ABB RobotStudio station: ABBRacer_20170305-223939.rsstn

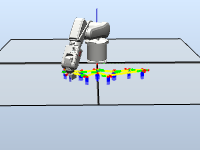
Station ABBRacer (saved by RobotStudio 6.4.7206.1027)
Controller IRB_120_3kg_0.58m, task T_ROB1: task frame (RAPID world) sits at (0, 0, 25) mm in the station
Controller IRB_120_3kg_0.58m
  mechanical unit ROB_1: IRB120_3_58__01, 6 joints, base frame (0, 0, 0) mm
Layout (positions relative to the parent item):
  - IRB120_3_58__01 [mechanism, from Robots\IRB120_3_58_G_01.rslib] at (0, 0, 25) mm; joint values [-0.4552, 1.5213, -0.5651, 0, 0.6146, 3.1228] (rad or m)
  - Bakje [part] at (432.53, -170.17, 50) mm, rotated rx -90 ry 0 rz 155 deg
Attachment: Bakje is attached to IRB120_3_58__01 / Link6
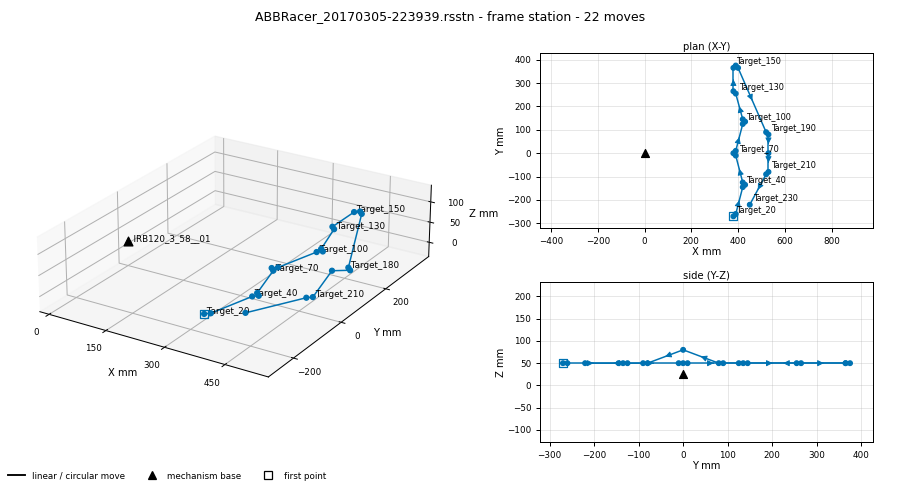
[picture p0: tool path of ABBRacer_20170305-223939.rsstn in frame station, 22 of 22 moves have a stored position in this frame; points joined in program order, loops and branches not executed]
Targets, tools, work objects and paths stored in the station, written as RAPID:
! task T_ROB1
MODULE Module1
  CONST robtarget Target_20:=[[380,-270,25],[0,0,1,0],[-1,0,-1,0],[9E+09,9E+09,9E+09,9E+09,9E+09,9E+09]];
  CONST robtarget Target_30:=[[390,-260,25],[0,0.130526192,0.991444861,0],[-1,-1,-1,0],[9E+09,9E+09,9E+09,9E+09,9E+09,9E+09]];
  CONST robtarget Target_40:=[[420,-145,25],[0,0.258819045,0.965925826,0],[-1,0,-1,0],[9E+09,9E+09,9E+09,9E+09,9E+09,9E+09]];
  CONST robtarget Target_50:=[[430.000232033,-134.999844259,25.000157187],[0.00000015,0,1,-0.000000047],[-1,0,-1,0],[9E+09,9E+09,9E+09,9E+09,9E+09,9E+09]];
  CONST robtarget Target_60:=[[420,-125,25],[0,-0.130526192,0.991444861,0],[-1,0,-1,0],[9E+09,9E+09,9E+09,9E+09,9E+09,9E+09]];
  CONST robtarget Target_70:=[[390,-10,25],[0,-0.3007058,0.953716951,0],[-1,-1,-1,0],[9E+09,9E+09,9E+09,9E+09,9E+09,9E+09]];
  CONST robtarget Target_80:=[[380.000012735,0,25.000038681],[0.000000135,0,1,0],[0,0,0,0],[9E+09,9E+09,9E+09,9E+09,9E+09,9E+09]];
  CONST robtarget Target_90:=[[390,10,25],[0,0.130526192,0.991444861,0],[0,0,0,0],[9E+09,9E+09,9E+09,9E+09,9E+09,9E+09]];
  CONST robtarget Target_100:=[[420,125,25],[0,0.3007058,0.953716951,0],[0,-1,0,0],[9E+09,9E+09,9E+09,9E+09,9E+09,9E+09]];
  CONST robtarget Target_110:=[[430,135,25],[0,0,1,0],[0,-1,0,0],[9E+09,9E+09,9E+09,9E+09,9E+09,9E+09]];
  CONST robtarget Target_120:=[[420,145,25],[0,-0.130526192,0.991444861,0],[0,-1,0,0],[9E+09,9E+09,9E+09,9E+09,9E+09,9E+09]];
  CONST robtarget Target_130:=[[390,255,25],[0,-0.3007058,0.953716951,0],[0,0,0,0],[9E+09,9E+09,9E+09,9E+09,9E+09,9E+09]];
  CONST robtarget Target_140:=[[379.999778696,265.000063835,24.999829243],[-0.000000287,0,1,-0.0000002],[0,0,0,0],[9E+09,9E+09,9E+09,9E+09,9E+09,9E+09]];
  CONST robtarget Target_150:=[[380,365,25],[0,0.130526192,0.991444861,0],[0,0,0,0],[9E+09,9E+09,9E+09,9E+09,9E+09,9E+09]];
  CONST robtarget Target_160:=[[390,375,25],[0,0.707106781,0.707106781,0],[0,-1,0,0],[9E+09,9E+09,9E+09,9E+09,9E+09,9E+09]];
  CONST robtarget Target_170:=[[400,365,25],[0,0.976296007,0.216439614,0],[0,0,0,0],[9E+09,9E+09,9E+09,9E+09,9E+09,9E+09]];
  CONST robtarget Target_180:=[[520,90,25],[0,0.976296007,0.216439614,0],[0,0,0,0],[9E+09,9E+09,9E+09,9E+09,9E+09,9E+09]];
  CONST robtarget Target_190:=[[530,80,25],[0,1,0,0],[0,-1,1,0],[9E+09,9E+09,9E+09,9E+09,9E+09,9E+09]];
  CONST robtarget Target_200:=[[529.999952018,0,54.999958724],[0,1,-0.000000163,0.000000127],[0,-1,2,0],[9E+09,9E+09,9E+09,9E+09,9E+09,9E+09]];
  CONST robtarget Target_210:=[[530.000040299,-79.999757507,24.999982632],[0.000000023,1,0.000000306,0.000000155],[-1,0,1,0],[9E+09,9E+09,9E+09,9E+09,9E+09,9E+09]];
  CONST robtarget Target_220:=[[520.000978391,-90.0002022,25.001612523],[0.000000563,0.976296148,-0.216438979,0.00000269],[-1,-1,2,0],[9E+09,9E+09,9E+09,9E+09,9E+09,9E+09]];
  CONST robtarget Target_230:=[[449.999555293,-220.247787183,24.999520517],[-0.000000187,0.976295901,-0.216440094,-0.000000774],[-1,0,1,0],[9E+09,9E+09,9E+09,9E+09,9E+09,9E+09]];
  PROC Path_10()
    MoveL Target_20,v500,z50,tool0\WObj:=wobj0;
    MoveL Target_30,v500,z50,tool0\WObj:=wobj0;
    MoveL Target_40,v500,z50,tool0\WObj:=wobj0;
    MoveL Target_50,v500,z50,tool0\WObj:=wobj0;
    MoveL Target_60,v500,z50,tool0\WObj:=wobj0;
    MoveL Target_70,v500,z50,tool0\WObj:=wobj0;
    MoveL Target_80,v500,z50,tool0\WObj:=wobj0;
    MoveL Target_90,v500,z50,tool0\WObj:=wobj0;
    MoveL Target_100,v500,z50,tool0\WObj:=wobj0;
    MoveL Target_110,v500,z50,tool0\WObj:=wobj0;
    MoveL Target_120,v500,z50,tool0\WObj:=wobj0;
    MoveL Target_130,v500,z50,tool0\WObj:=wobj0;
    MoveL Target_140,v500,z50,tool0\WObj:=wobj0;
    MoveL Target_150,v500,z50,tool0\WObj:=wobj0;
    MoveL Target_160,v500,z50,tool0\WObj:=wobj0;
    MoveL Target_170,v500,z50,tool0\WObj:=wobj0;
    MoveL Target_180,v500,z50,tool0\WObj:=wobj0;
    MoveL Target_190,v500,z50,tool0\WObj:=wobj0;
    MoveL Target_200,v500,z50,tool0\WObj:=wobj0;
    MoveL Target_210,v500,z50,tool0\WObj:=wobj0;
    MoveL Target_220,v500,z50,tool0\WObj:=wobj0;
    MoveL Target_230,v500,z50,tool0\WObj:=wobj0;
  ENDPROC
ENDMODULE

